Staubli VAL3: Frame.dtx

bool bExit
bool bListRefresh
bool bUserRefresh
public frame fFrame{}
  [Frame1] = {x=480, y=190, z=-101.4, rx=2, rz=-90, fatherId=world[0]}
  [Frame10] = {fatherId=world[0]}
  [Frame11] = {fatherId=world[0]}
  [Frame12] = {fatherId=world[0]}
  [Frame13] = {fatherId=world[0]}
  [Frame14] = {fatherId=world[0]}
  [Frame15] = {fatherId=world[0]}
  [Frame16] = {fatherId=world[0]}
  [Frame17] = {fatherId=world[0]}
  [Frame18] = {fatherId=world[0]}
  [Frame19] = {fatherId=world[0]}
  [Frame2] = {fatherId=world[0]}
  [Frame20] = {fatherId=world[0]}
  [Frame3] = {fatherId=world[0]}
  [Frame4] = {fatherId=world[0]}
  [Frame5] = {fatherId=world[0]}
  [Frame6] = {fatherId=world[0]}
  [Frame7] = {fatherId=world[0]}
  [Frame8] = {fatherId=world[0]}
  [Frame9] = {fatherId=world[0]}
mdesc mNomSpeed
num nSelected
num nType
string sFrameName
string sItem
string sList
string sListItemValue
string sParameter
